(* Logix 5000 project; controller STAT 1756-L72 rev 20.12; software revision 20.04; part 26 of 34 *)
(* tags used below, declared in another part *)
   B3 : DINT[35];
   F8 : REAL[100];
   N20 : DINT[50];
   N7 : DINT[150];
   N9 : DINT[200];
   S : INT[164];
   T4 : TIMER[100];
   ibtlancy1 : DINT;
   mwcsth : DINT;
   mwcsthh : DINT;
   mwcstl : DINT;
   mwcstll : DINT;
   N11 : DINT[150];
   S_FLOW_VENTURI : DINT;
   s_flw_filtrat_flt_presse : REAL;
   s_hac_turbidity : REAL;
   s_lvl_buffert_flt_presse : REAL;
   s_lvl_filtraat_water_from_flt : DINT;
   s_lvl_holding_tk : REAL;
   s_lvl_lift_tk : REAL;
   s_lvl_Ph_bac : REAL;
   s_lvl_puisard_L123 : REAL;
   s_lvl_reacteur_lancy : REAL;
   s_optek_turbidity : REAL;
   s_pos_V_filtrat : REAL;
   scp_flw_filtrat_flt_presse : SCP;
   scp_hac_turbidity : SCP;
   scp_lvl_buffer_flt_presse : SCP;
   scp_lvl_filtraat_water_from_flt : SCP;
   scp_lvl_holding_tk : SCP;
   scp_lvl_lift_tk : SCP;
   scp_lvl_Ph_bac : SCP;
   scp_lvl_puisard_L123 : SCP;
   scp_lvl_reacteur_lancy : SCP;
   scp_optek_turbidity : SCP;
   scp_pos_V_filtrat : SCP;
   vanne_filtraaT : REAL;
(* LANCY, continued *)

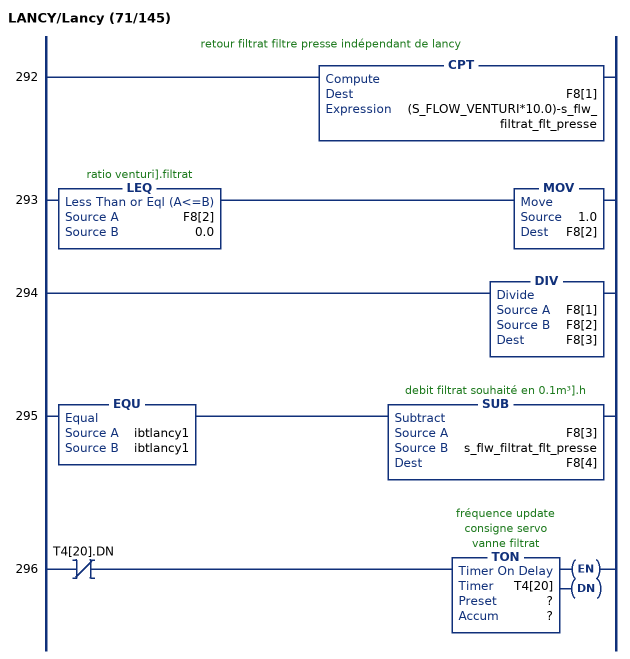
   // retour filtrat filtre presse indépendant de lancy
   292: CPT(F8[1],(S_FLOW_VENTURI*10.0)-s_flw_filtrat_flt_presse);
   293: LEQ(F8[2],0.0)MOV(1.0,F8[2]);
   294: DIV(F8[1],F8[2],F8[3]);
   295: EQU(ibtlancy1,ibtlancy1)SUB(F8[3],s_flw_filtrat_flt_presse,F8[4]);
   296: XIO(T4[20].DN)TON(T4[20],?,?);
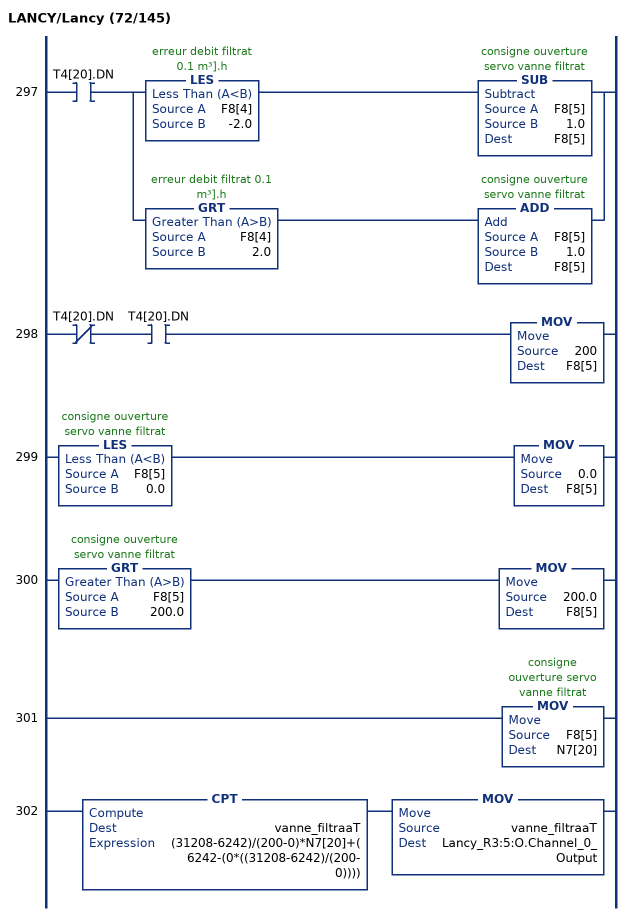
   297: XIC(T4[20].DN)[LES(F8[4],-2.0) SUB(F8[5],1.0,F8[5]) ,GRT(F8[4],2.0) ADD(F8[5],1.0,F8[5]) ];
   298: XIO(T4[20].DN)XIC(T4[20].DN)MOV(200,F8[5]);
   299: LES(F8[5],0.0)MOV(0.0,F8[5]);
   300: GRT(F8[5],200.0)MOV(200.0,F8[5]);
   301: MOV(F8[5],N7[20]);
   302: CPT(vanne_filtraaT,(31208-6242)/(200-0)*N7[20]+(6242-(0*((31208-6242)/(200-0)))))MOV(vanne_filtraaT,Lancy_R3:5:O.Channel_0_Output);
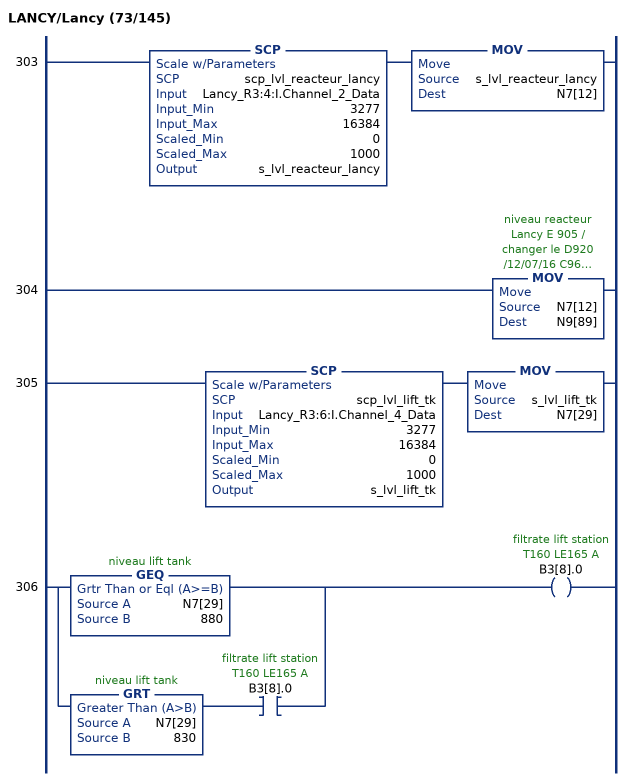
   303: SCP(scp_lvl_reacteur_lancy,Lancy_R3:4:I.Channel_2_Data,3277,16384,0,1000,s_lvl_reacteur_lancy)MOV(s_lvl_reacteur_lancy,N7[12]);
   304: MOV(N7[12],N9[89]);
   305: SCP(scp_lvl_lift_tk,Lancy_R3:6:I.Channel_4_Data,3277,16384,0,1000,s_lvl_lift_tk)MOV(s_lvl_lift_tk,N7[29]);
   306: [GEQ(N7[29],880) ,GRT(N7[29],830) XIC(B3[8].0) ]OTE(B3[8].0);
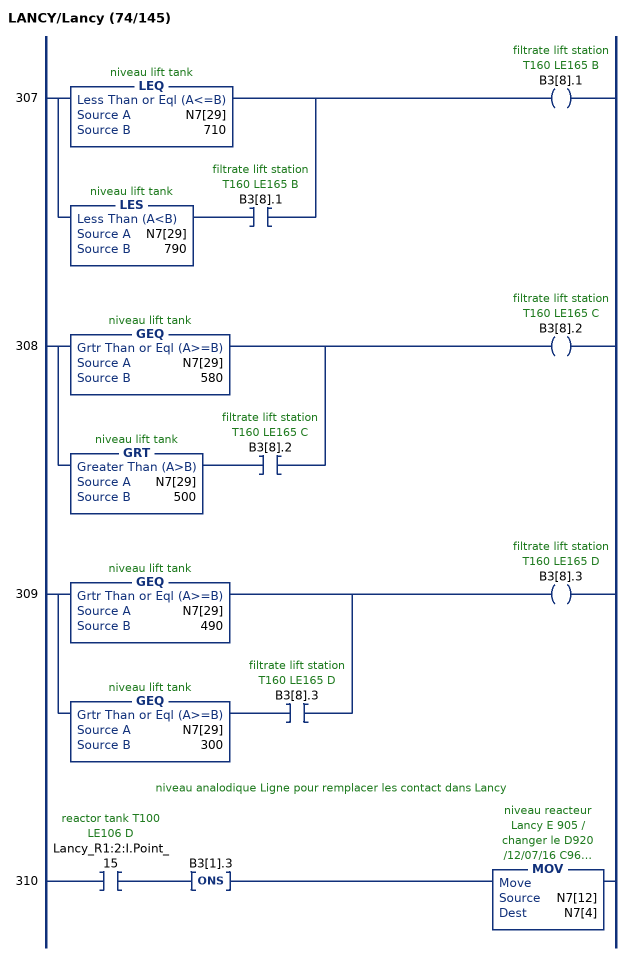
   307: [LEQ(N7[29],710) ,LES(N7[29],790) XIC(B3[8].1) ]OTE(B3[8].1);
   308: [GEQ(N7[29],580) ,GRT(N7[29],500) XIC(B3[8].2) ]OTE(B3[8].2);
   309: [GEQ(N7[29],490) ,GEQ(N7[29],300) XIC(B3[8].3) ]OTE(B3[8].3);
   // niveau analodique Ligne pour remplacer les contact dans Lancy
   310: XIC(Lancy_R1:2:I.Point_15)ONS(B3[1].3)MOV(N7[12],N7[4]);
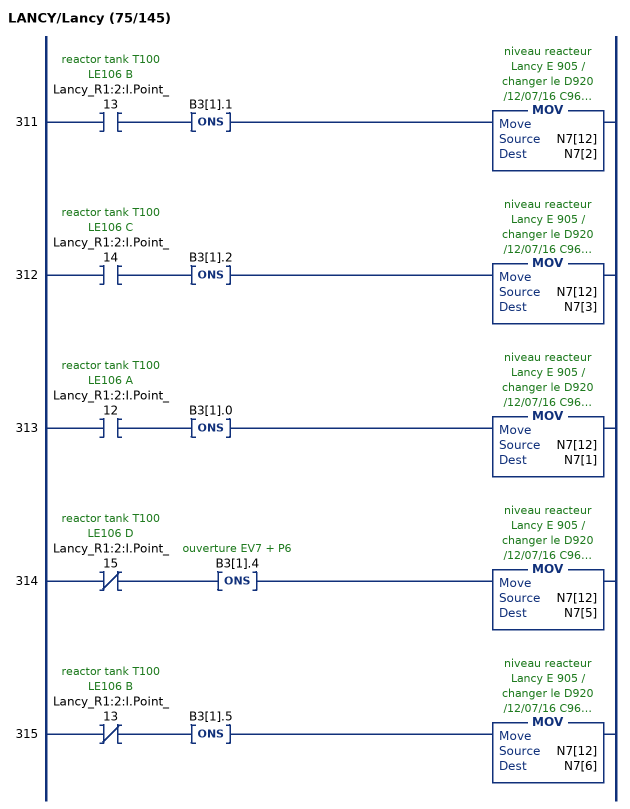
   311: XIC(Lancy_R1:2:I.Point_13)ONS(B3[1].1)MOV(N7[12],N7[2]);
   312: XIC(Lancy_R1:2:I.Point_14)ONS(B3[1].2)MOV(N7[12],N7[3]);
   313: XIC(Lancy_R1:2:I.Point_12)ONS(B3[1].0)MOV(N7[12],N7[1]);
   314: XIO(Lancy_R1:2:I.Point_15)ONS(B3[1].4)MOV(N7[12],N7[5]);
   315: XIO(Lancy_R1:2:I.Point_13)ONS(B3[1].5)MOV(N7[12],N7[6]);
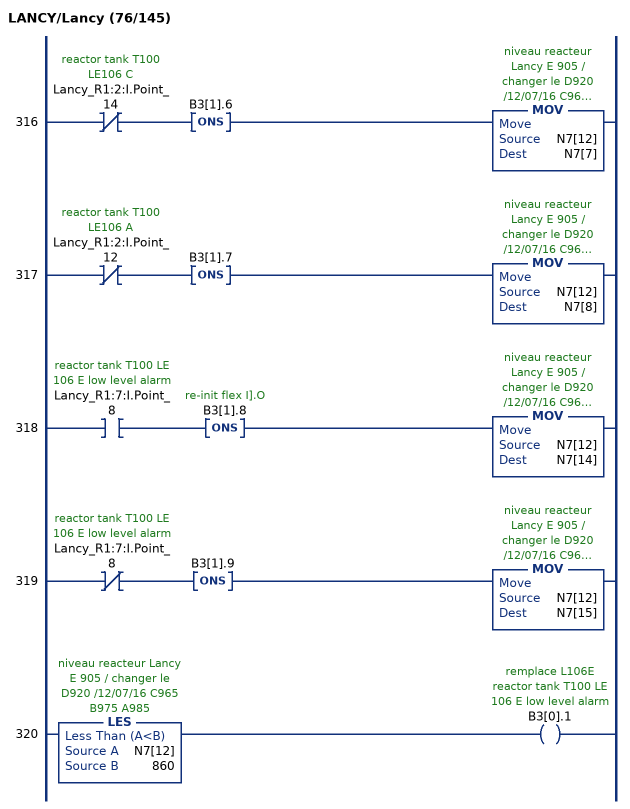
   316: XIO(Lancy_R1:2:I.Point_14)ONS(B3[1].6)MOV(N7[12],N7[7]);
   317: XIO(Lancy_R1:2:I.Point_12)ONS(B3[1].7)MOV(N7[12],N7[8]);
   318: XIC(Lancy_R1:7:I.Point_8)ONS(B3[1].8)MOV(N7[12],N7[14]);
   319: XIO(Lancy_R1:7:I.Point_8)ONS(B3[1].9)MOV(N7[12],N7[15]);
   320: LES(N7[12],860)OTE(B3[0].1);
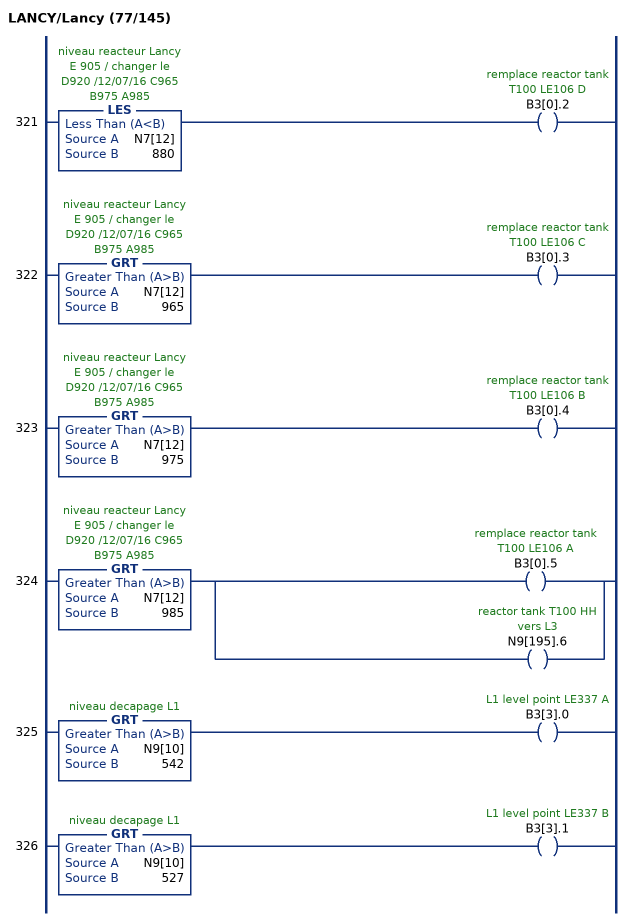
   321: LES(N7[12],880)OTE(B3[0].2);
   322: GRT(N7[12],965)OTE(B3[0].3);
   323: GRT(N7[12],975)OTE(B3[0].4);
   324: GRT(N7[12],985)[OTE(B3[0].5) ,OTE(N9[195].6) ];
   325: GRT(N9[10],542)OTE(B3[3].0);
   326: GRT(N9[10],527)OTE(B3[3].1);
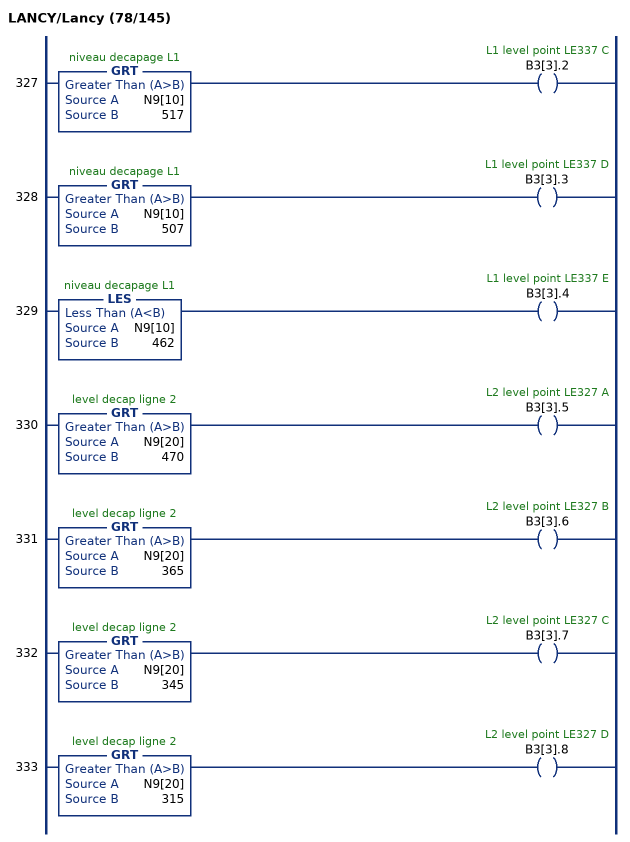
   327: GRT(N9[10],517)OTE(B3[3].2);
   328: GRT(N9[10],507)OTE(B3[3].3);
   329: LES(N9[10],462)OTE(B3[3].4);
   330: GRT(N9[20],470)OTE(B3[3].5);
   331: GRT(N9[20],365)OTE(B3[3].6);
   332: GRT(N9[20],345)OTE(B3[3].7);
   333: GRT(N9[20],315)OTE(B3[3].8);
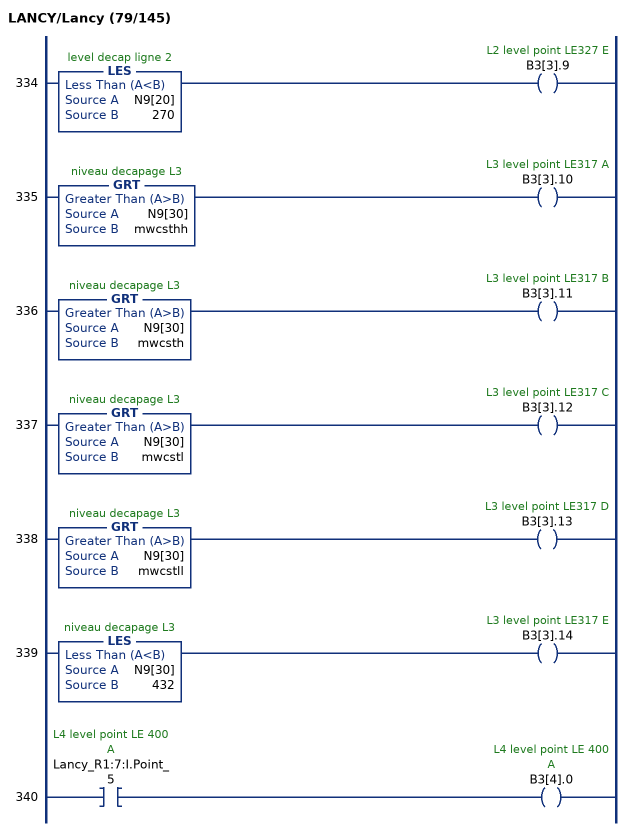
   334: LES(N9[20],270)OTE(B3[3].9);
   335: GRT(N9[30],mwcsthh)OTE(B3[3].10);
   336: GRT(N9[30],mwcsth)OTE(B3[3].11);
   337: GRT(N9[30],mwcstl)OTE(B3[3].12);
   338: GRT(N9[30],mwcstll)OTE(B3[3].13);
   339: LES(N9[30],432)OTE(B3[3].14);
   340: XIC(Lancy_R1:7:I.Point_5)OTE(B3[4].0);
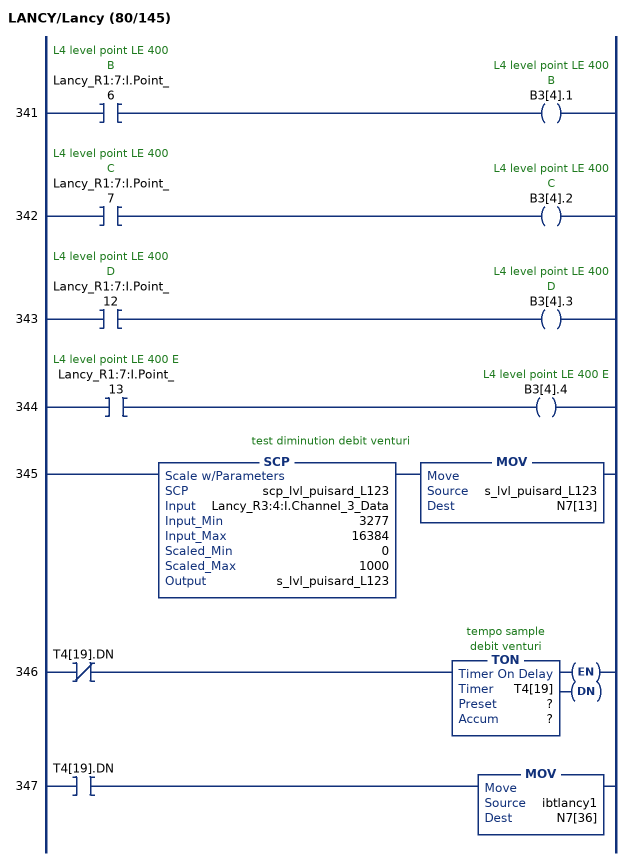
   341: XIC(Lancy_R1:7:I.Point_6)OTE(B3[4].1);
   342: XIC(Lancy_R1:7:I.Point_7)OTE(B3[4].2);
   343: XIC(Lancy_R1:7:I.Point_12)OTE(B3[4].3);
   344: XIC(Lancy_R1:7:I.Point_13)OTE(B3[4].4);
   // test diminution debit venturi
   345: SCP(scp_lvl_puisard_L123,Lancy_R3:4:I.Channel_3_Data,3277,16384,0,1000,s_lvl_puisard_L123)MOV(s_lvl_puisard_L123,N7[13]);
   346: XIO(T4[19].DN)TON(T4[19],?,?);
   347: XIC(T4[19].DN)MOV(ibtlancy1,N7[36]);
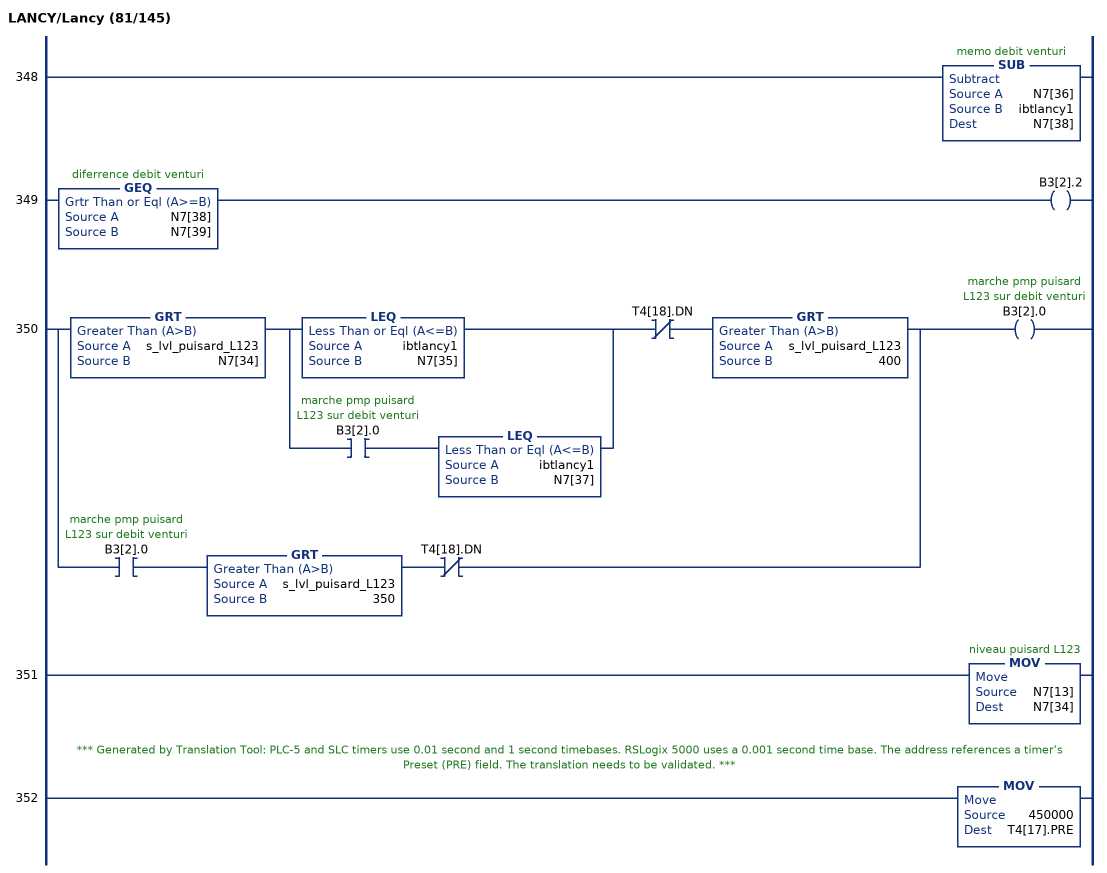
   348: SUB(N7[36],ibtlancy1,N7[38]);
   349: GEQ(N7[38],N7[39])OTE(B3[2].2);
   350: [GRT(s_lvl_puisard_L123,N7[34]) [LEQ(ibtlancy1,N7[35]) ,XIC(B3[2].0) LEQ(ibtlancy1,N7[37]) ] XIO(T4[18].DN) GRT(s_lvl_puisard_L123,400) ,XIC(B3[2].0) GRT(s_lvl_puisard_L123,350) XIO(T4[18].DN) ]OTE(B3[2].0);
   351: MOV(N7[13],N7[34]);
   // *** Generated by Translation Tool: PLC-5 and SLC timers use 0.01 second and 1 second timebases. RSLogix 5000 uses a 0.001 second time base. The address references a timer’s Preset (PRE) field. The translation needs to be validated. ***
   352: MOV(450000,T4[17].PRE);
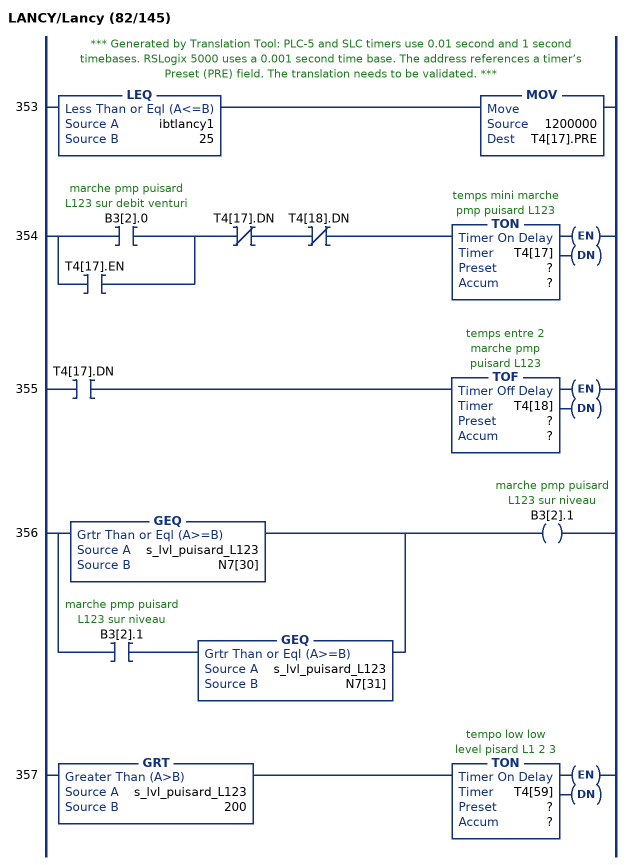
   // *** Generated by Translation Tool: PLC-5 and SLC timers use 0.01 second and 1 second timebases. RSLogix 5000 uses a 0.001 second time base. The address references a timer’s Preset (PRE) field. The translation needs to be validated. ***
   353: LEQ(ibtlancy1,25)MOV(1200000,T4[17].PRE);
   354: [XIC(B3[2].0) ,XIC(T4[17].EN) ]XIO(T4[17].DN)XIO(T4[18].DN)TON(T4[17],?,?);
   355: XIC(T4[17].DN)TOF(T4[18],?,?);
   356: [GEQ(s_lvl_puisard_L123,N7[30]) ,XIC(B3[2].1) GEQ(s_lvl_puisard_L123,N7[31]) ]OTE(B3[2].1);
   357: GRT(s_lvl_puisard_L123,200)TON(T4[59],?,?);
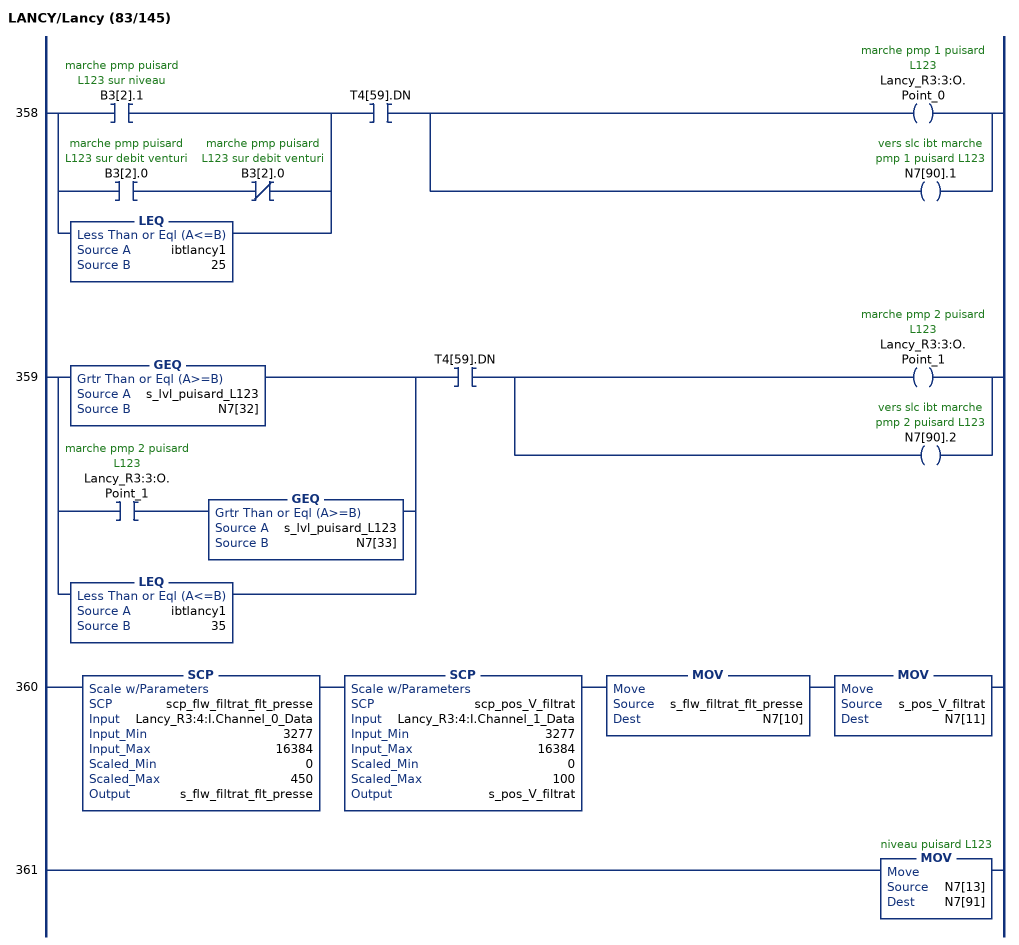
   358: [XIC(B3[2].1) ,XIC(B3[2].0) XIO(B3[2].0) ,LEQ(ibtlancy1,25) ]XIC(T4[59].DN)[OTE(Lancy_R3:3:O.Point_0) ,OTE(N7[90].1) ];
   359: [GEQ(s_lvl_puisard_L123,N7[32]) ,XIC(Lancy_R3:3:O.Point_1) GEQ(s_lvl_puisard_L123,N7[33]) ,LEQ(ibtlancy1,35) ]XIC(T4[59].DN)[OTE(Lancy_R3:3:O.Point_1) ,OTE(N7[90].2) ];
   360: SCP(scp_flw_filtrat_flt_presse,Lancy_R3:4:I.Channel_0_Data,3277,16384,0,450,s_flw_filtrat_flt_presse)SCP(scp_pos_V_filtrat,Lancy_R3:4:I.Channel_1_Data,3277,16384,0,100,s_pos_V_filtrat)MOV(s_flw_filtrat_flt_presse,N7[10])MOV(s_pos_V_filtrat,N7[11]);
   361: MOV(N7[13],N7[91]);
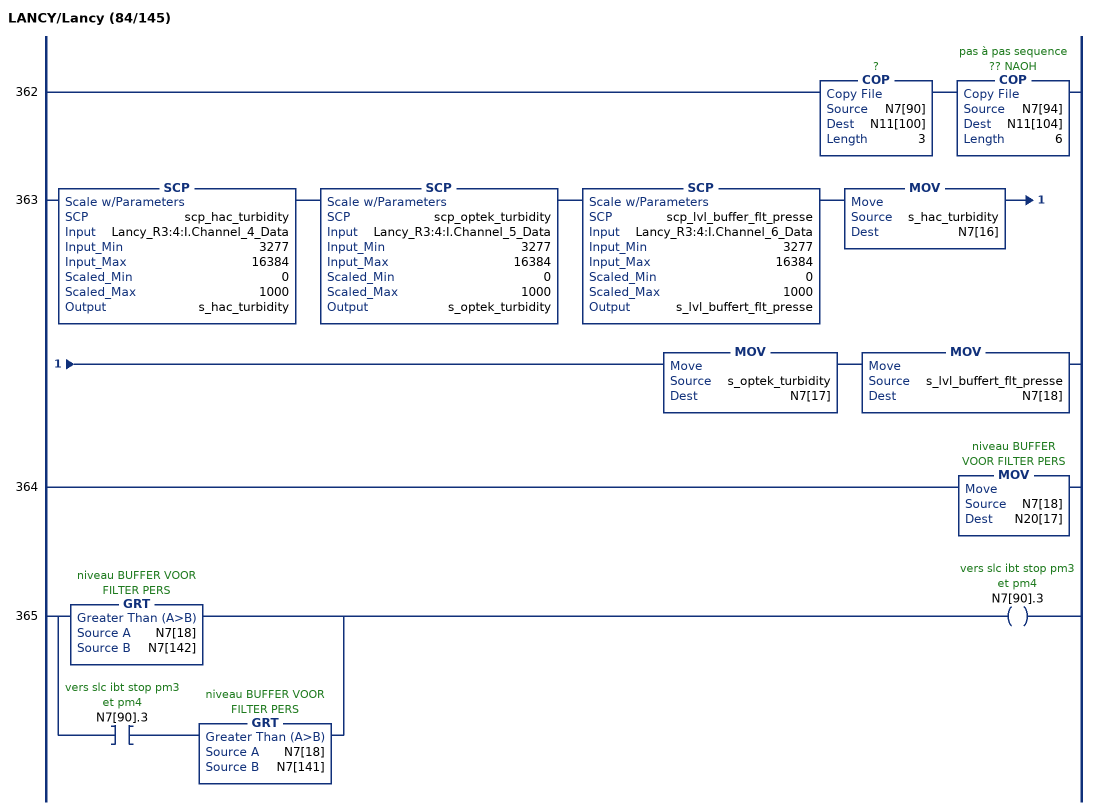
   362: COP(N7[90],N11[100],3)COP(N7[94],N11[104],6);
   363: SCP(scp_hac_turbidity,Lancy_R3:4:I.Channel_4_Data,3277,16384,0,1000,s_hac_turbidity)SCP(scp_optek_turbidity,Lancy_R3:4:I.Channel_5_Data,3277,16384,0,1000,s_optek_turbidity)SCP(scp_lvl_buffer_flt_presse,Lancy_R3:4:I.Channel_6_Data,3277,16384,0,1000,s_lvl_buffert_flt_presse)MOV(s_hac_turbidity,N7[16])MOV(s_optek_turbidity,N7[17])MOV(s_lvl_buffert_flt_presse,N7[18]);
   364: MOV(N7[18],N20[17]);
   365: [GRT(N7[18],N7[142]) ,XIC(N7[90].3) GRT(N7[18],N7[141]) ]OTE(N7[90].3);
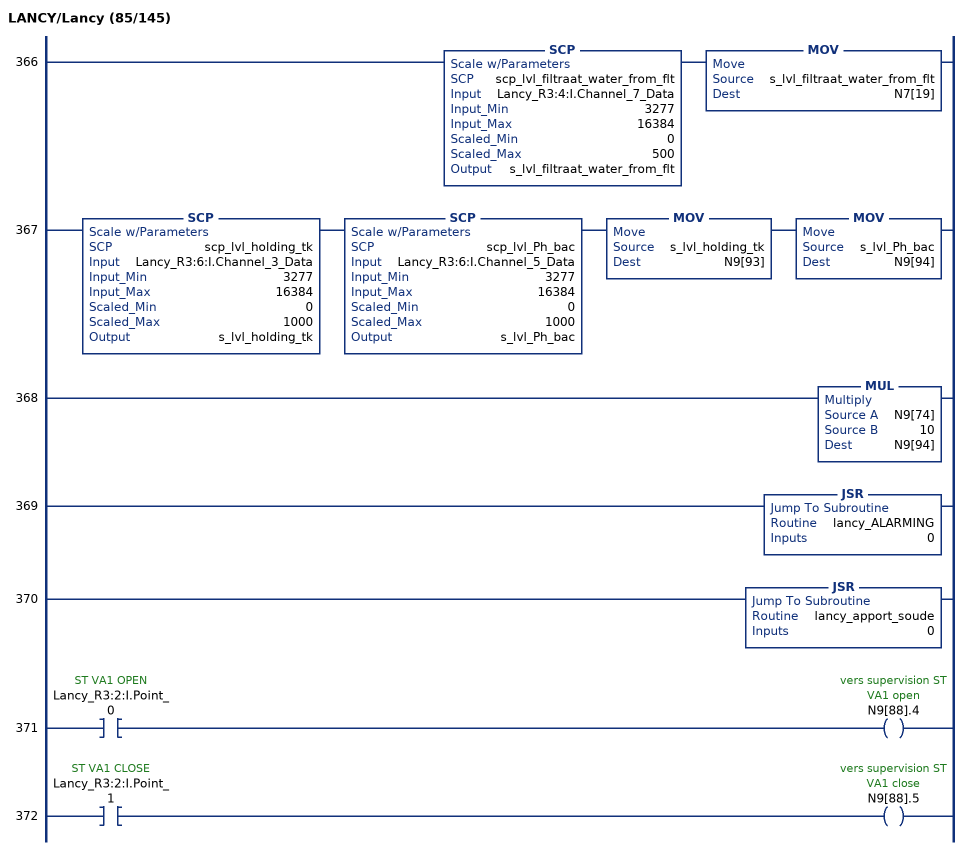
   366: SCP(scp_lvl_filtraat_water_from_flt,Lancy_R3:4:I.Channel_7_Data,3277,16384,0,500,s_lvl_filtraat_water_from_flt)MOV(s_lvl_filtraat_water_from_flt,N7[19]);
   367: SCP(scp_lvl_holding_tk,Lancy_R3:6:I.Channel_3_Data,3277,16384,0,1000,s_lvl_holding_tk)SCP(scp_lvl_Ph_bac,Lancy_R3:6:I.Channel_5_Data,3277,16384,0,1000,s_lvl_Ph_bac)MOV(s_lvl_holding_tk,N9[93])MOV(s_lvl_Ph_bac,N9[94]);
   368: MUL(N9[74],10,N9[94]);
   369: JSR(lancy_ALARMING,0);
   370: JSR(lancy_apport_soude,0);
   371: XIC(Lancy_R3:2:I.Point_0)OTE(N9[88].4);
   372: XIC(Lancy_R3:2:I.Point_1)OTE(N9[88].5);
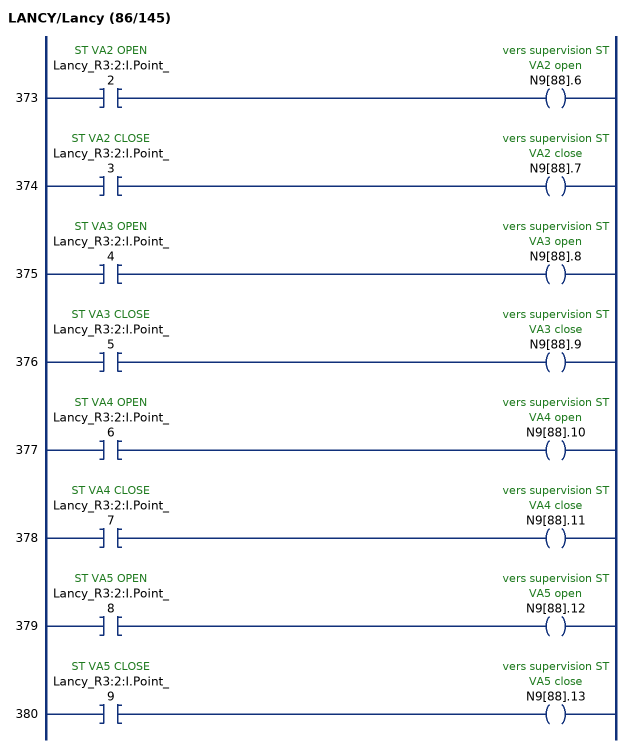
   373: XIC(Lancy_R3:2:I.Point_2)OTE(N9[88].6);
   374: XIC(Lancy_R3:2:I.Point_3)OTE(N9[88].7);
   375: XIC(Lancy_R3:2:I.Point_4)OTE(N9[88].8);
   376: XIC(Lancy_R3:2:I.Point_5)OTE(N9[88].9);
   377: XIC(Lancy_R3:2:I.Point_6)OTE(N9[88].10);
   378: XIC(Lancy_R3:2:I.Point_7)OTE(N9[88].11);
   379: XIC(Lancy_R3:2:I.Point_8)OTE(N9[88].12);
   380: XIC(Lancy_R3:2:I.Point_9)OTE(N9[88].13);
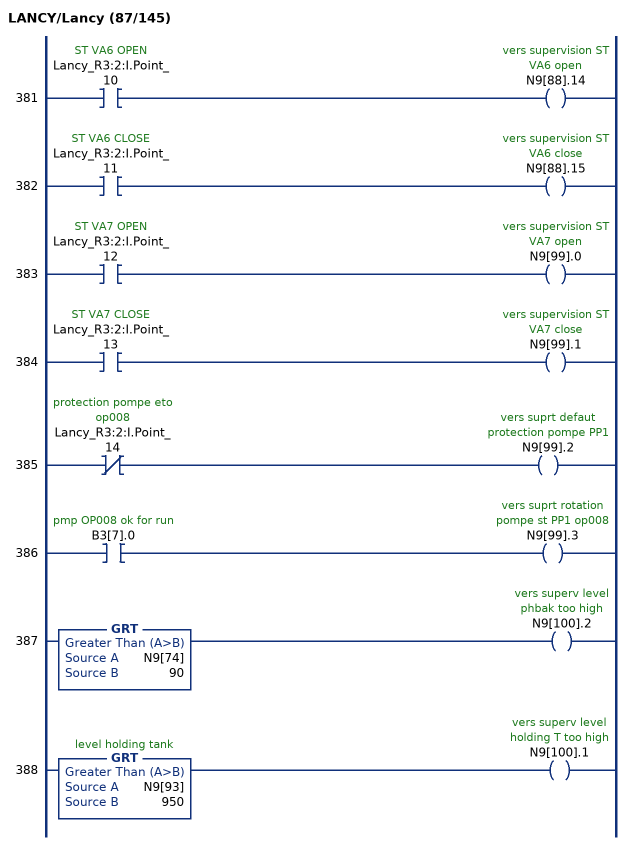
   381: XIC(Lancy_R3:2:I.Point_10)OTE(N9[88].14);
   382: XIC(Lancy_R3:2:I.Point_11)OTE(N9[88].15);
   383: XIC(Lancy_R3:2:I.Point_12)OTE(N9[99].0);
   384: XIC(Lancy_R3:2:I.Point_13)OTE(N9[99].1);
   385: XIO(Lancy_R3:2:I.Point_14)OTE(N9[99].2);
   386: XIC(B3[7].0)OTE(N9[99].3);
   387: GRT(N9[74],90)OTE(N9[100].2);
   388: GRT(N9[93],950)OTE(N9[100].1);
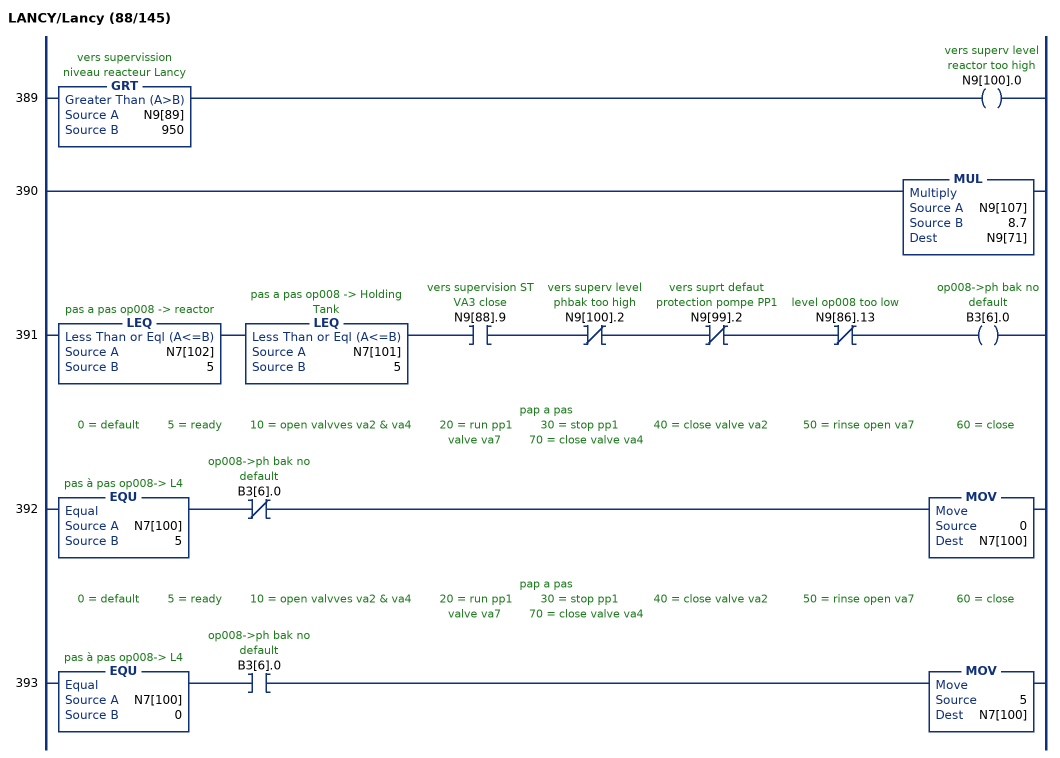
   389: GRT(N9[89],950)OTE(N9[100].0);
   390: MUL(N9[107],8.7,N9[71]);
   391: LEQ(N7[102],5)LEQ(N7[101],5)XIC(N9[88].9)XIO(N9[100].2)XIO(N9[99].2)XIO(N9[86].13)OTE(B3[6].0);
   // pap a pas
   // 0 = default        5 = ready        10 = open valvves va2 & va4        20 = run pp1        30 = stop pp1          40 = close valve va2          50 = rinse open va7            60 = close valve va7        70 = close valve va4
   392: EQU(N7[100],5)XIO(B3[6].0)MOV(0,N7[100]);
   // pap a pas
   // 0 = default        5 = ready        10 = open valvves va2 & va4        20 = run pp1        30 = stop pp1          40 = close valve va2          50 = rinse open va7            60 = close valve va7        70 = close valve va4
   393: EQU(N7[100],0)XIC(B3[6].0)MOV(5,N7[100]);
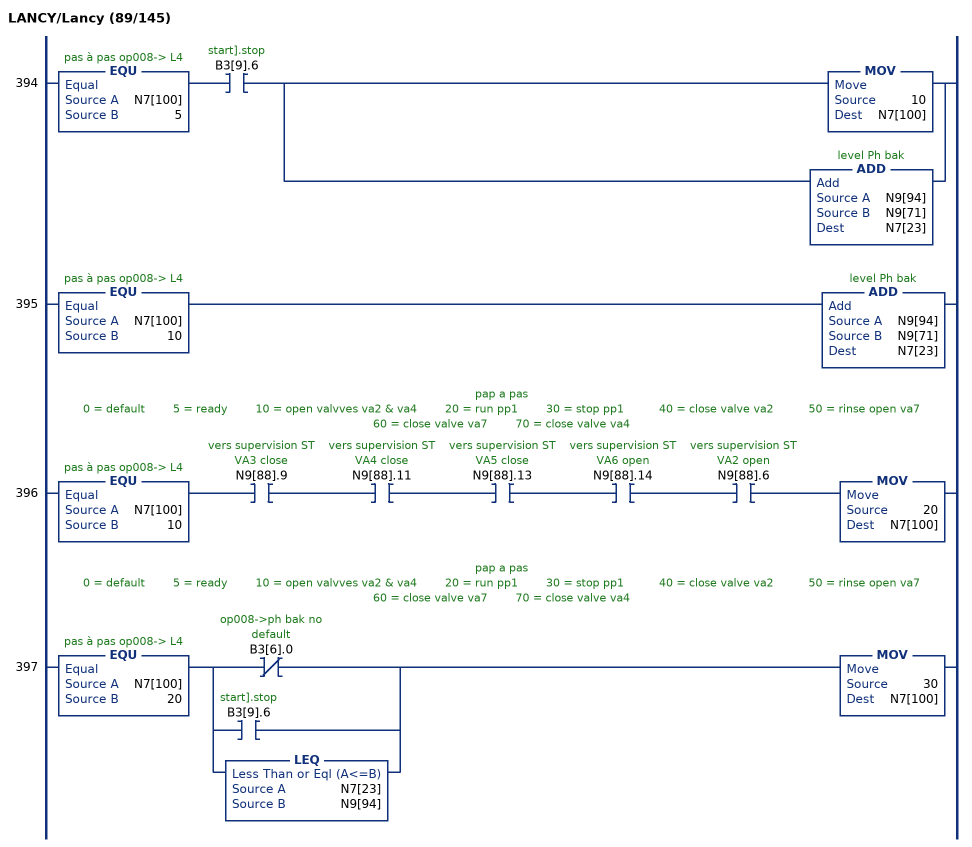
   394: EQU(N7[100],5)XIC(B3[9].6)[MOV(10,N7[100]) ,ADD(N9[94],N9[71],N7[23]) ];
   395: EQU(N7[100],10)ADD(N9[94],N9[71],N7[23]);
   // pap a pas
   // 0 = default        5 = ready        10 = open valvves va2 & va4        20 = run pp1        30 = stop pp1          40 = close valve va2          50 = rinse open va7            60 = close valve va7        70 = close valve va4
   396: EQU(N7[100],10)XIC(N9[88].9)XIC(N9[88].11)XIC(N9[88].13)XIC(N9[88].14)XIC(N9[88].6)MOV(20,N7[100]);
   // pap a pas
   // 0 = default        5 = ready        10 = open valvves va2 & va4        20 = run pp1        30 = stop pp1          40 = close valve va2          50 = rinse open va7            60 = close valve va7        70 = close valve va4
   397: EQU(N7[100],20)[XIO(B3[6].0) ,XIC(B3[9].6) ,LEQ(N7[23],N9[94]) ]MOV(30,N7[100]);
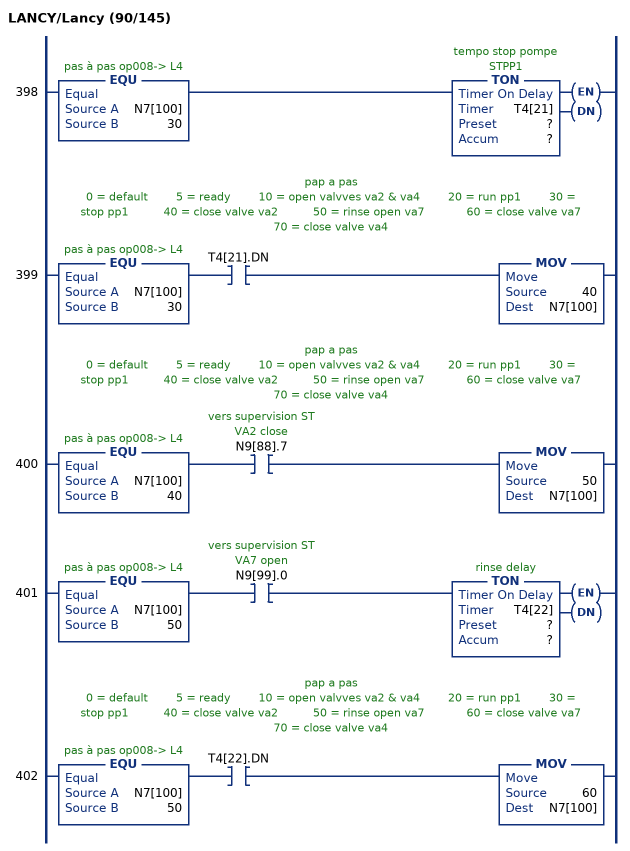
   398: EQU(N7[100],30)TON(T4[21],?,?);
   // pap a pas
   // 0 = default        5 = ready        10 = open valvves va2 & va4        20 = run pp1        30 = stop pp1          40 = close valve va2          50 = rinse open va7            60 = close valve va7        70 = close valve va4
   399: EQU(N7[100],30)XIC(T4[21].DN)MOV(40,N7[100]);
   // pap a pas
   // 0 = default        5 = ready        10 = open valvves va2 & va4        20 = run pp1        30 = stop pp1          40 = close valve va2          50 = rinse open va7            60 = close valve va7        70 = close valve va4
   400: EQU(N7[100],40)XIC(N9[88].7)MOV(50,N7[100]);
   401: EQU(N7[100],50)XIC(N9[99].0)TON(T4[22],?,?);
   // pap a pas
   // 0 = default        5 = ready        10 = open valvves va2 & va4        20 = run pp1        30 = stop pp1          40 = close valve va2          50 = rinse open va7            60 = close valve va7        70 = close valve va4
   402: EQU(N7[100],50)XIC(T4[22].DN)MOV(60,N7[100]);
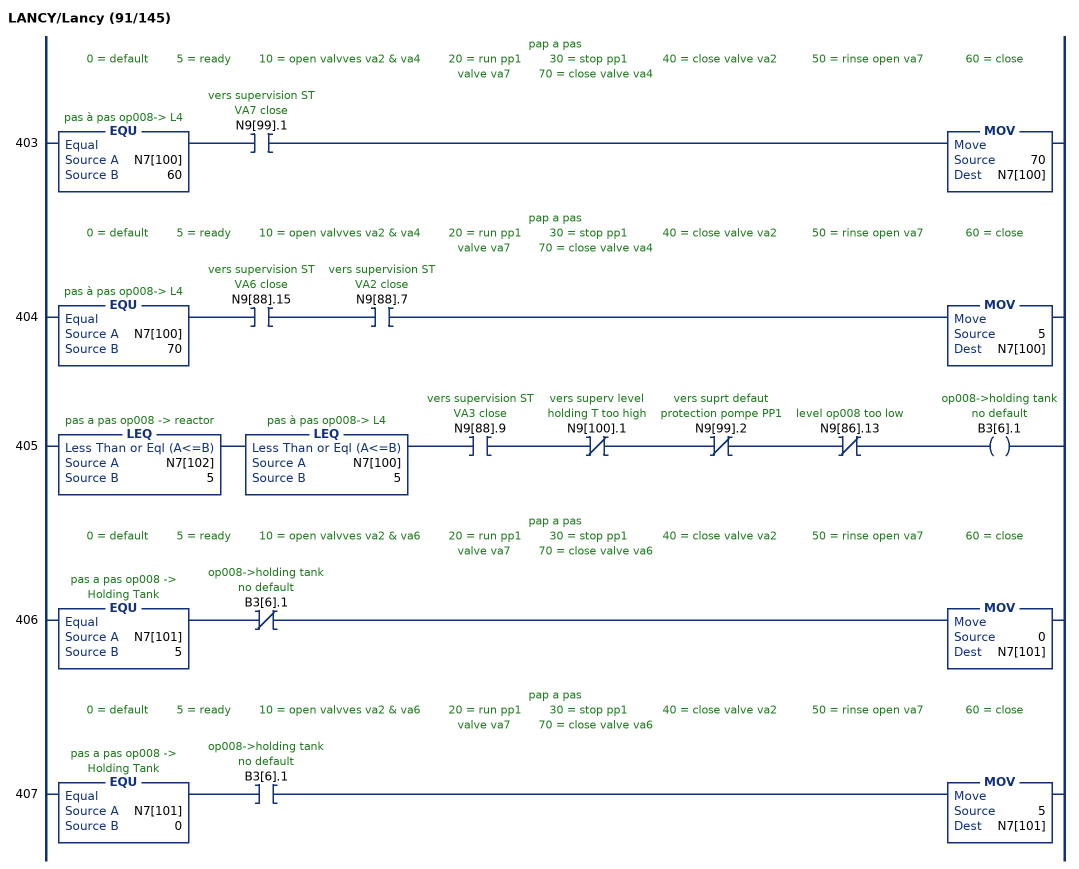
   // pap a pas
   // 0 = default        5 = ready        10 = open valvves va2 & va4        20 = run pp1        30 = stop pp1          40 = close valve va2          50 = rinse open va7            60 = close valve va7        70 = close valve va4
   403: EQU(N7[100],60)XIC(N9[99].1)MOV(70,N7[100]);
   // pap a pas
   // 0 = default        5 = ready        10 = open valvves va2 & va4        20 = run pp1        30 = stop pp1          40 = close valve va2          50 = rinse open va7            60 = close valve va7        70 = close valve va4
   404: EQU(N7[100],70)XIC(N9[88].15)XIC(N9[88].7)MOV(5,N7[100]);
   405: LEQ(N7[102],5)LEQ(N7[100],5)XIC(N9[88].9)XIO(N9[100].1)XIO(N9[99].2)XIO(N9[86].13)OTE(B3[6].1);
   // pap a pas
   // 0 = default        5 = ready        10 = open valvves va2 & va6        20 = run pp1        30 = stop pp1          40 = close valve va2          50 = rinse open va7            60 = close valve va7        70 = close valve va6
   406: EQU(N7[101],5)XIO(B3[6].1)MOV(0,N7[101]);
   // pap a pas
   // 0 = default        5 = ready        10 = open valvves va2 & va6        20 = run pp1        30 = stop pp1          40 = close valve va2          50 = rinse open va7            60 = close valve va7        70 = close valve va6
   407: EQU(N7[101],0)XIC(B3[6].1)MOV(5,N7[101]);
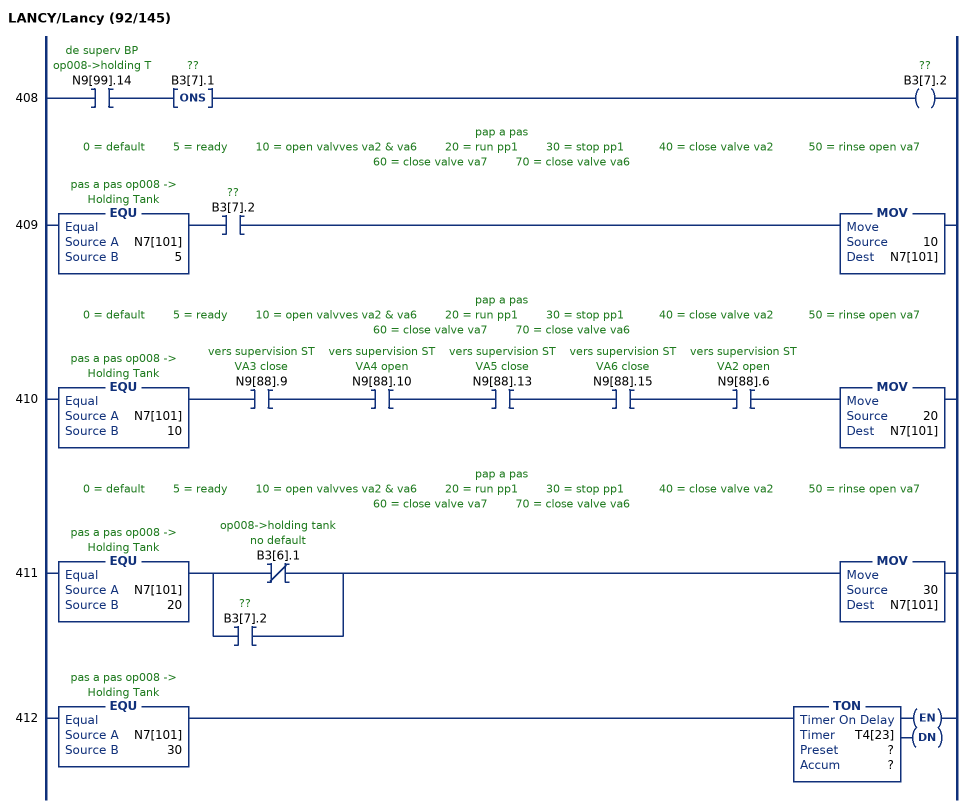
   408: XIC(N9[99].14)ONS(B3[7].1)OTE(B3[7].2);
   // pap a pas
   // 0 = default        5 = ready        10 = open valvves va2 & va6        20 = run pp1        30 = stop pp1          40 = close valve va2          50 = rinse open va7            60 = close valve va7        70 = close valve va6
   409: EQU(N7[101],5)XIC(B3[7].2)MOV(10,N7[101]);
   // pap a pas
   // 0 = default        5 = ready        10 = open valvves va2 & va6        20 = run pp1        30 = stop pp1          40 = close valve va2          50 = rinse open va7            60 = close valve va7        70 = close valve va6
   410: EQU(N7[101],10)XIC(N9[88].9)XIC(N9[88].10)XIC(N9[88].13)XIC(N9[88].15)XIC(N9[88].6)MOV(20,N7[101]);
   // pap a pas
   // 0 = default        5 = ready        10 = open valvves va2 & va6        20 = run pp1        30 = stop pp1          40 = close valve va2          50 = rinse open va7            60 = close valve va7        70 = close valve va6
   411: EQU(N7[101],20)[XIO(B3[6].1) ,XIC(B3[7].2) ]MOV(30,N7[101]);
   412: EQU(N7[101],30)TON(T4[23],?,?);
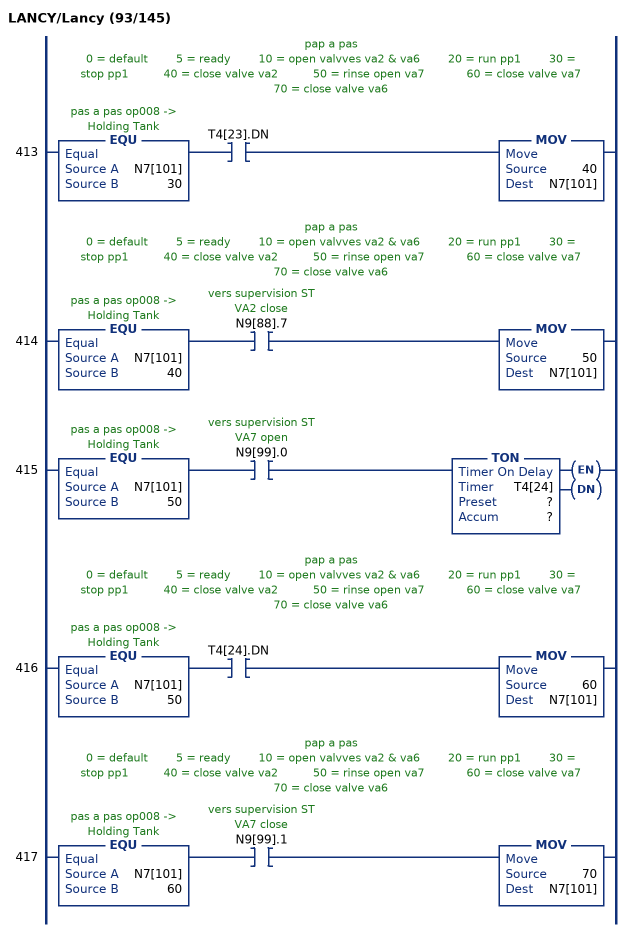
   // pap a pas
   // 0 = default        5 = ready        10 = open valvves va2 & va6        20 = run pp1        30 = stop pp1          40 = close valve va2          50 = rinse open va7            60 = close valve va7        70 = close valve va6
   413: EQU(N7[101],30)XIC(T4[23].DN)MOV(40,N7[101]);
   // pap a pas
   // 0 = default        5 = ready        10 = open valvves va2 & va6        20 = run pp1        30 = stop pp1          40 = close valve va2          50 = rinse open va7            60 = close valve va7        70 = close valve va6
   414: EQU(N7[101],40)XIC(N9[88].7)MOV(50,N7[101]);
   415: EQU(N7[101],50)XIC(N9[99].0)TON(T4[24],?,?);
   // pap a pas
   // 0 = default        5 = ready        10 = open valvves va2 & va6        20 = run pp1        30 = stop pp1          40 = close valve va2          50 = rinse open va7            60 = close valve va7        70 = close valve va6
   416: EQU(N7[101],50)XIC(T4[24].DN)MOV(60,N7[101]);
   // pap a pas
   // 0 = default        5 = ready        10 = open valvves va2 & va6        20 = run pp1        30 = stop pp1          40 = close valve va2          50 = rinse open va7            60 = close valve va7        70 = close valve va6
   417: EQU(N7[101],60)XIC(N9[99].1)MOV(70,N7[101]);
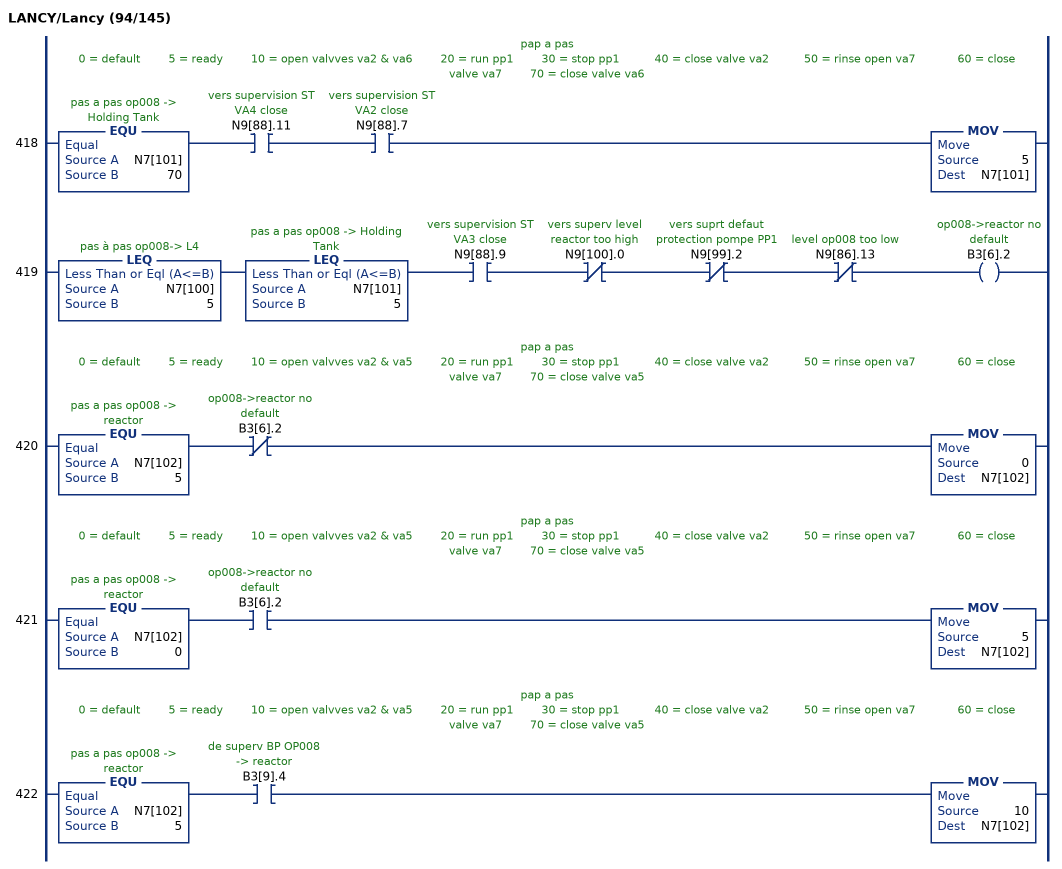
   // pap a pas
   // 0 = default        5 = ready        10 = open valvves va2 & va6        20 = run pp1        30 = stop pp1          40 = close valve va2          50 = rinse open va7            60 = close valve va7        70 = close valve va6
   418: EQU(N7[101],70)XIC(N9[88].11)XIC(N9[88].7)MOV(5,N7[101]);
   419: LEQ(N7[100],5)LEQ(N7[101],5)XIC(N9[88].9)XIO(N9[100].0)XIO(N9[99].2)XIO(N9[86].13)OTE(B3[6].2);
   // pap a pas
   // 0 = default        5 = ready        10 = open valvves va2 & va5        20 = run pp1        30 = stop pp1          40 = close valve va2          50 = rinse open va7            60 = close valve va7        70 = close valve va5
   420: EQU(N7[102],5)XIO(B3[6].2)MOV(0,N7[102]);
   // pap a pas
   // 0 = default        5 = ready        10 = open valvves va2 & va5        20 = run pp1        30 = stop pp1          40 = close valve va2          50 = rinse open va7            60 = close valve va7        70 = close valve va5
   421: EQU(N7[102],0)XIC(B3[6].2)MOV(5,N7[102]);
   // pap a pas
   // 0 = default        5 = ready        10 = open valvves va2 & va5        20 = run pp1        30 = stop pp1          40 = close valve va2          50 = rinse open va7            60 = close valve va7        70 = close valve va5
   422: EQU(N7[102],5)XIC(B3[9].4)MOV(10,N7[102]);
